# EPICS autosave request: iocBoot/iocUSB3104/auto_settings.req
file "USB3104_settings.req", P=$(P)
